(*
An abstract representation of a system state, providing the foundation for implementing state-specific behavior.  
Manages its owner entity and supports state transitions within the system.  
Offers default behavior for state lifecycle methods, allowing programmers to override only the relevant parts.
*)
FUNCTION_BLOCK ABSTRACT State IMPLEMENTS I_StateInternal, I_State
VAR
	{attribute 'hide'}
	_comp						: Component(THIS^);
	{attribute 'hide'}
	_bInQueue					: BOOL;
	{attribute 'hide'}
	_iNextInBuffer				: I_StateInternal; // State Buffer management
	
	_tag			: TagBase;	
END_VAR

PROPERTY INTERNAL FINAL _AsIState : I_State
GET
_AsIState := THIS^;
END_GET
END_PROPERTY

PROPERTY INTERNAL FINAL _AsIStateInternal : I_StateInternal
GET
_AsIStateInternal := THIS^;
END_GET
END_PROPERTY

METHOD INTERNAL _CanActivate : BOOL
_CanActivate := CanActivate();
END_METHOD

METHOD INTERNAL _CanDeactivate : BOOL
_CanDeactivate := CanDeactivate();
END_METHOD

PROPERTY INTERNAL _InQueue : BOOL
GET
_InQueue := _bInQueue;
END_GET
SET
_bInQueue := _InQueue;
END_SET
END_PROPERTY

PROPERTY INTERNAL _NextInBuffer : I_StateInternal
GET
_NextInBuffer := _iNextInBuffer;
END_GET
SET
_iNextInBuffer := _NextInBuffer;
END_SET
END_PROPERTY

METHOD INTERNAL _OnEntry
OnEntry();
END_METHOD

METHOD INTERNAL _OnExecute
OnExecute();
END_METHOD

METHOD INTERNAL _OnExit
OnExit();
END_METHOD

(*
Determines whether the state can be activated.  
Returns `TRUE` by default but can be overridden for specific activation conditions.
*)
METHOD PROTECTED CanActivate : BOOL
VAR_INPUT
END_VAR
CanActivate := TRUE;
END_METHOD

(*
Determines whether the state can be deactivated.  
Returns `TRUE` by default but can be overridden for specific deactivation conditions.
*)
METHOD PROTECTED CanDeactivate : BOOL
VAR_INPUT
END_VAR
CanDeactivate := TRUE;
END_METHOD

//FB_Init is always available implicitly and it is used primarily for initialization.
//The return value is not evaluated. For a specific influence, you can also declare the
//methods explicitly and provide additional code there with the standard initialization
//code. You can evaluate the return value.
{attribute 'hide'}
METHOD FB_Init: BOOL
VAR_INPUT
    bInitRetains: BOOL; // TRUE: the retain variables are initialized (reset warm / reset cold)
    bInCopyCode: BOOL;  // TRUE: the instance will be copied to the copy code afterward (online change)   
END_VAR
END_METHOD

(*
Executed when the state is entered.  
Provides a hook for defining state-specific behavior to be performed during the transition into this state.
*)
METHOD PROTECTED OnEntry
VAR_INPUT
END_VAR
END_METHOD

(*
Executed during the state's operation.  
Used to define state-specific logic that runs while the state is active.
*)
METHOD PROTECTED OnExecute
VAR_INPUT
END_VAR
END_METHOD

(*
Executed when the state transitions to another state.  
Provides a hook for defining cleanup or transition-specific behavior.
*)
METHOD PROTECTED OnExit
VAR_INPUT
END_VAR
END_METHOD

(*
Returns the entity that owns this state.
*)
PROPERTY FINAL Owner : I_Entity
GET
Owner := _comp.Entity;
END_GET
END_PROPERTY

(*
Allows initializing an external interface variable with an interface pointer to this instance within declaration block.
Example:
iState: I_State;
state: SomeState := (Proxy := iState);
Result: iState <> 0 
*)
PROPERTY Proxy : REFERENCE TO I_State
SET
Proxy := THIS^;
END_SET
END_PROPERTY

(*
Provides access to the `I_Tag` associated with the state.
*)
PROPERTY FINAL Tag : I_Tag
GET
Tag := _tag;
END_GET
END_PROPERTY

END_FUNCTION_BLOCK

(* stored: Version 1.1.0.1
   POU State: Id {a3b28716-f684-494e-889b-84fe1781ad45}, SpecialFunc None
   Folder _: Id {b2082cde-a72a-48d1-bf2b-bfe685440ba0}
   Folder Can: Id {012b303c-ee19-4d59-a8c5-29d7ee56e39c}
   Folder On: Id {5034b126-7af1-4e3e-aa65-10d454bc5f51}
   Property _AsIState: Id {ae988e03-7493-46d9-85de-be6948de1d8e}
   Get Get: Id {4c9d6b0d-006b-455b-828d-2ce5937584f8}
   Property _AsIStateInternal: Id {4fe75cff-cf53-4cef-a5a6-8ca77becdd1c}
   Get Get: Id {d8d590d5-9436-40ea-add0-78eaf9a46d23}
   Method _CanActivate: Id {71c49a83-838e-4656-9fc2-ce8957b8e198}
   Method _CanDeactivate: Id {d9ac8857-b429-40a0-ae64-2f200213bb6e}
   Property _InQueue: Id {00343d62-1ac6-4b7a-af5a-8983a284ec4e}
   Get Get: Id {ebe10328-99fb-4c92-9263-ffe964414865}
   Set Set: Id {fca23d48-8c9e-42f8-85fc-1b0cbdcaf6be}
   Property _NextInBuffer: Id {26c35362-4f86-4013-add5-ec59f766ab26}
   Get Get: Id {ef5ee735-cf5d-4c75-809d-088832acb881}
   Set Set: Id {798fc338-1046-4b35-b906-4ac80e5a26a0}
   Method _OnEntry: Id {233f0cb7-a018-4a8e-a04c-cd20357f448f}
   Method _OnExecute: Id {aabb82b9-2f5d-4e99-b353-6c10e3d6ce3d}
   Method _OnExit: Id {25d7c89a-22df-4af1-9c2c-e2be2f3e48a9}
   Method CanActivate: Id {dd755635-2c1b-4d2f-832c-8fe84230e7c4}
   Method CanDeactivate: Id {7b012b92-459d-4244-99c6-c8d2e693b887}
   Method FB_Init: Id {0426a892-c538-4afe-92f1-9f241d1ee74d}
   Method OnEntry: Id {71184392-1093-4315-9a73-835d846ab945}
   Method OnExecute: Id {1a4db232-f3d2-440c-9d63-b8a4efc99401}
   Method OnExit: Id {9584048f-886b-4757-b0ed-688b849511a2}
   Property Owner: Id {32b502a4-ba25-4a78-8e46-5a8b31e2a3e9}
   Get Get: Id {98a99666-df4c-40b9-abec-3c308e3cdead}
   Property Proxy: Id {e148912a-ec6c-4d53-987e-2cc3081d8267}
   Set Set: Id {c3e00474-819c-47ac-8733-a728d746c29b}
   Property Tag: Id {0bbeba40-ec6e-4b6d-a33f-9c84eca9c89e}
   Get Get: Id {c1b1ddfd-4e01-4e44-9d81-1a59ffd92985} *)
